// TIA Portal V17 export
// export: Created 2026-04-13T11:12:44.4548664Z, ExportSetting WithDefaults, DisplayName Totally Integrated Automation Portal, DisplayVersion V17 Update 4, DisplayName TIA Portal Openness, DisplayVersion V17 Update 4, DisplayName TIA Portal Version Control Interface, DisplayVersion V17, DisplayName SINAMICS Startdrive Advanced, DisplayVersion V17, DisplayName SINAMICS Startdrive G130, G150, S120, S150, SINAMICS MV, S210, DisplayVersion V17, DisplayName SINAMICS Startdrive G110M, G120, G120C, G120D, G120P, G115D, DisplayVersion V17, DisplayName STEP 7 Professional, DisplayVersion V17 Update 4, DisplayName STEP 7 Safety, DisplayVersion V17, DisplayName WinCC Professional, DisplayVersion V17 Update 4
DATA_BLOCK "A1-阀带反馈_DB"   // DB1
VERSION : 0.1
// stored: AutoNumber true, DBAccessibleFromOPCUA true, DBAccessibleFromWebserver true, InstanceOfName A1-阀带反馈, InstanceOfType FB
"A1-阀带反馈"
   // VAR
   //    泄压阀 { S7_SetPoint := 'True'} : "A3-普通阀控制";
   //    进风冷却水阀 { S7_SetPoint := 'True'} : "A3-普通阀控制";
   //    输送进风阀 { S7_SetPoint := 'True'} : "A3-普通阀控制";
   //    气流雾化阀 { S7_SetPoint := 'True'} : "A3-普通阀控制";
   //    开式排风隔断阀 { S7_SetPoint := 'True'} : "A3-普通阀控制";
   //    闭式排风隔断阀 { S7_SetPoint := 'True'} : "A3-普通阀控制";
   //    开式进风隔断阀 { S7_SetPoint := 'True'} : "A3-普通阀控制";
   //    闭式进风隔断阀 { S7_SetPoint := 'True'} : "A3-普通阀控制";
   //    一级冷却水阀 { S7_SetPoint := 'True'} : "A3-普通阀控制";
   //    二级冷冻水阀 { S7_SetPoint := 'True'} : "A3-普通阀控制";
   //    一级排液阀 { S7_SetPoint := 'True'} : "A3-普通阀控制";
   //    二级排液阀 { S7_SetPoint := 'True'} : "A3-普通阀控制";
   //    除雾排液阀 { S7_SetPoint := 'True'} : "A3-普通阀控制";
   //    补氮阀 : "A3-普通阀控制";
   //    进氮阀 { S7_SetPoint := 'True'} : "A3-普通阀控制";
   //    塔顶清洗球阀 { S7_SetPoint := 'True'} : "A3-普通阀控制";
   //    溶剂回收排放阀 { S7_SetPoint := 'True'} : "A3-普通阀控制";
   //    室内排水隔膜泵 { S7_SetPoint := 'True'} : "A3-普通阀控制";
   //    溶剂排液泵 { S7_SetPoint := 'True'} : "A3-普通阀控制";
   //    清洗伸缩气缸 { S7_SetPoint := 'True'} : "A3-普通阀控制";
   // END_VAR
BEGIN
END_DATA_BLOCK
